PROGRAM counterMaintenance
VAR
END_VAR

//Checks all of the sensors and resets the counter appropriatley as a maintenance check

IF Glbl.northStraightSensor = FALSE AND Glbl.southStraightSensor = FALSE THEN
	Glbl.state1Counter := 0;
	Glbl.northStraightSensorCnt := 0;
	Glbl.southStraightSensorCnt := 0;
END_IF

IF Glbl.eastStraightSensor = FALSE AND Glbl.westStraightSensor = FALSE THEN
	Glbl.state2Counter := 0;
	Glbl.eastStraightSensorCnt := 0;
	Glbl.westStraightSensorCnt := 0;
END_IF

IF Glbl.northLeftSensor = FALSE AND Glbl.southLeftSensor = FALSE THEN
	Glbl.state3Counter := 0;
	Glbl.northLeftSensorCnt := 0;
	Glbl.southLeftSensorCnt := 0;
END_IF

IF Glbl.eastLeftSensor = FALSE AND Glbl.westLeftSensor = FALSE THEN
	Glbl.state4Counter := 0;
	Glbl.eastLeftSensorCnt := 0;
	Glbl.westLeftSensorCnt := 0;
END_IF

IF Glbl.northStraightSensor = FALSE AND Glbl.northLeftSensor = FALSE THEN
	Glbl.state5Counter := 0;
	Glbl.northStraightSensorCnt := 0;
	Glbl.northLeftSensorCnt := 0;
END_IF

IF Glbl.southStraightSensor = FALSE AND Glbl.southLeftSensor = FALSE THEN
	Glbl.state6Counter := 0;
	Glbl.southStraightSensorCnt := 0;
	Glbl.southLeftSensorCnt := 0;
END_IF

IF Glbl.eastStraightSensor = FALSE AND Glbl.eastLeftSensor = FALSE THEN
	Glbl.state7Counter := 0;
	Glbl.eastStraightSensorCnt := 0;
	Glbl.eastLeftSensorCnt := 0;
END_IF

IF Glbl.westStraightSensor = FALSE AND Glbl.westLeftSensor = FALSE THEN
	Glbl.state8Counter := 0;
	Glbl.westStraightSensorCnt := 0;
	Glbl.westLeftSensorCnt := 0;
END_IF

END_PROGRAM

(* stored: Version 1.1.0.1, ProductVersion 3.1.4022.10
   POU counterMaintenance: Id {5902e63f-7fb3-4abb-a307-2501c204c8e9}, SpecialFunc None *)
